// Mitsubishi GX Works2 project: plctest   PLC: Q02/Q02H

PROGRAM MAIN
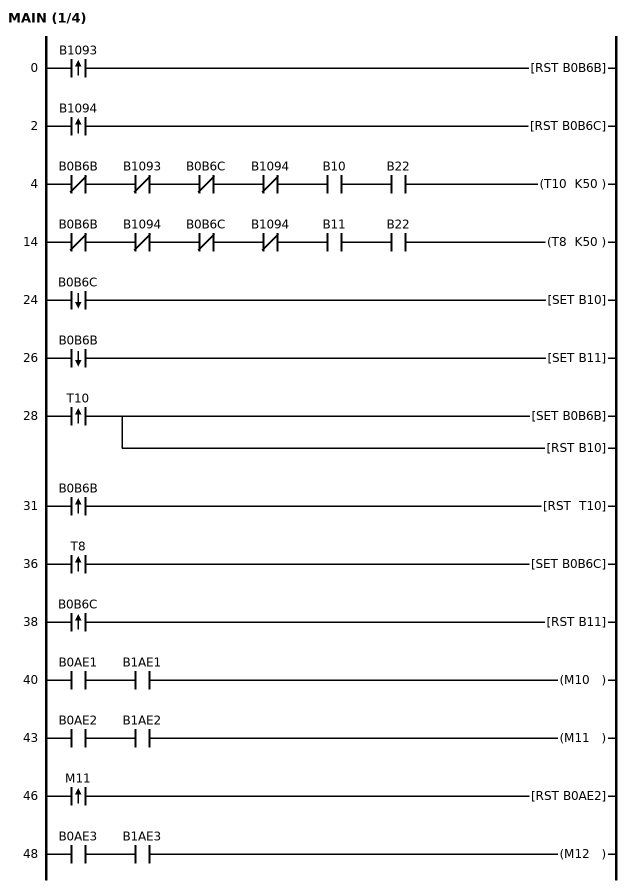
0     LDP     B1093
      RST     B0B6B
2     LDP     B1094
      RST     B0B6C
4     LDI     B0B6B
      ANI     B1093
      ANI     B0B6C
      ANI     B1094
      AND     B10
      AND     B22
      OUT     T10 K50
14    LDI     B0B6B
      ANI     B1094
      ANI     B0B6C
      ANI     B1094
      AND     B11
      AND     B22
      OUT     T8 K50
24    LDF     B0B6C
      SET     B10
26    LDF     B0B6B
      SET     B11
28    LDP     T10
      SET     B0B6B
      RST     B10
31    LDP     B0B6B
      RST     T10
36    LDP     T8
      SET     B0B6C
38    LDP     B0B6C
      RST     B11
40    LD      B0AE1
      AND     B1AE1
      OUT     M10
43    LD      B0AE2
      AND     B1AE2
      OUT     M11
46    LDP     M11
      RST     B0AE2
48    LD      B0AE3
      AND     B1AE3
      OUT     M12
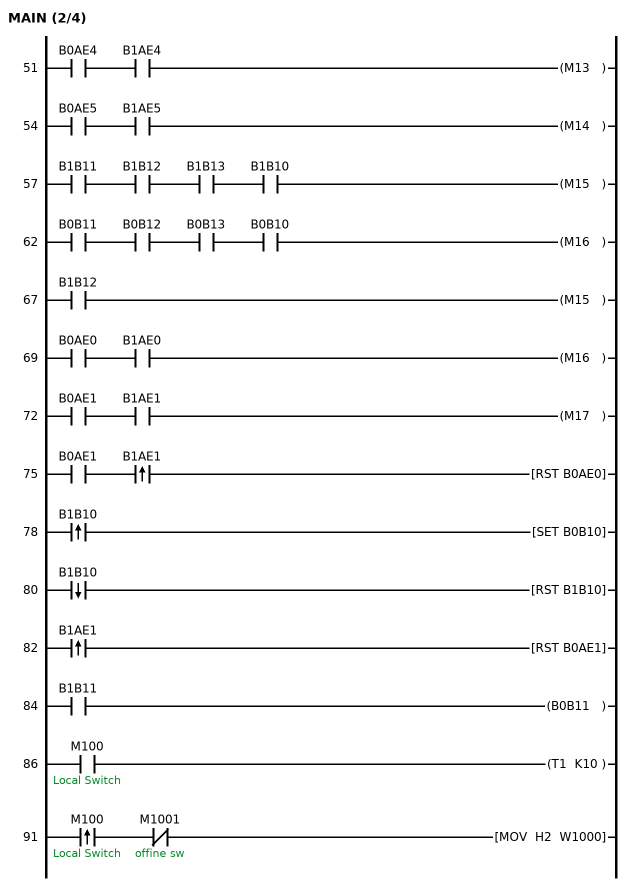
51    LD      B0AE4
      AND     B1AE4
      OUT     M13
54    LD      B0AE5
      AND     B1AE5
      OUT     M14
57    LD      B1B11
      AND     B1B12
      AND     B1B13
      AND     B1B10
      OUT     M15
62    LD      B0B11
      AND     B0B12
      AND     B0B13
      AND     B0B10
      OUT     M16
67    LD      B1B12
      OUT     M15
69    LD      B0AE0
      AND     B1AE0
      OUT     M16
72    LD      B0AE1
      AND     B1AE1
      OUT     M17
75    LD      B0AE1
      ANDP    B1AE1
      RST     B0AE0
78    LDP     B1B10
      SET     B0B10
80    LDF     B1B10
      RST     B1B10
82    LDP     B1AE1
      RST     B0AE1
84    LD      B1B11
      OUT     B0B11
86    LD      M100  ; Local Switch
      OUT     T1 K10
91    LDP     M100  ; Local Switch
      ANI     M1001  ; offine sw
      MOV     H2 W1000
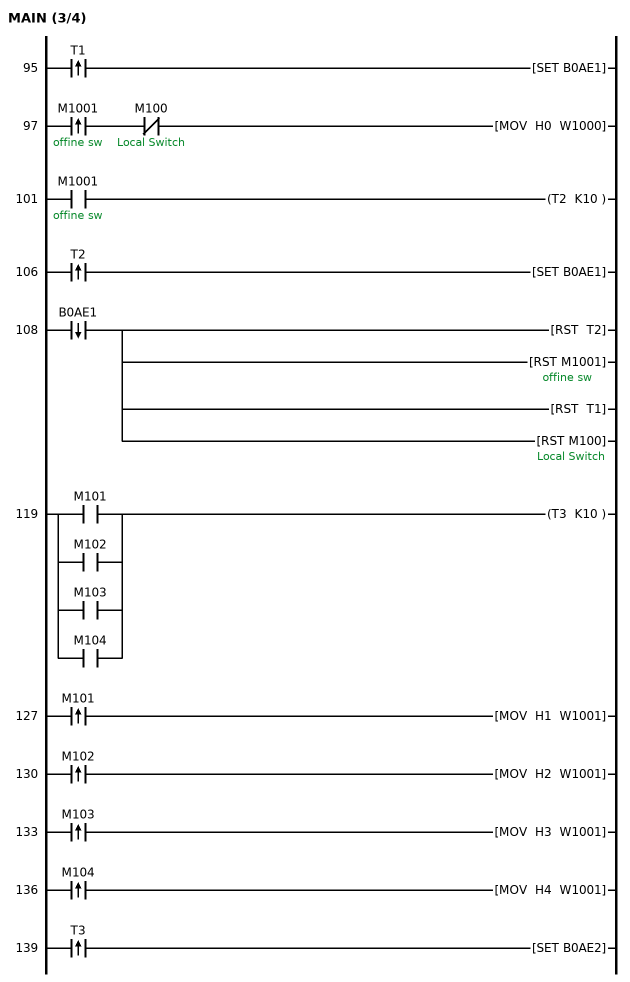
95    LDP     T1
      SET     B0AE1
97    LDP     M1001  ; offine sw
      ANI     M100  ; Local Switch
      MOV     H0 W1000
101   LD      M1001  ; offine sw
      OUT     T2 K10
106   LDP     T2
      SET     B0AE1
108   LDF     B0AE1
      RST     T2
      RST     M1001  ; offine sw
      RST     T1
      RST     M100  ; Local Switch
119   LD      M101
      OR      M102
      OR      M103
      OR      M104
      OUT     T3 K10
127   LDP     M101
      MOV     H1 W1001
130   LDP     M102
      MOV     H2 W1001
133   LDP     M103
      MOV     H3 W1001
136   LDP     M104
      MOV     H4 W1001
139   LDP     T3
      SET     B0AE2
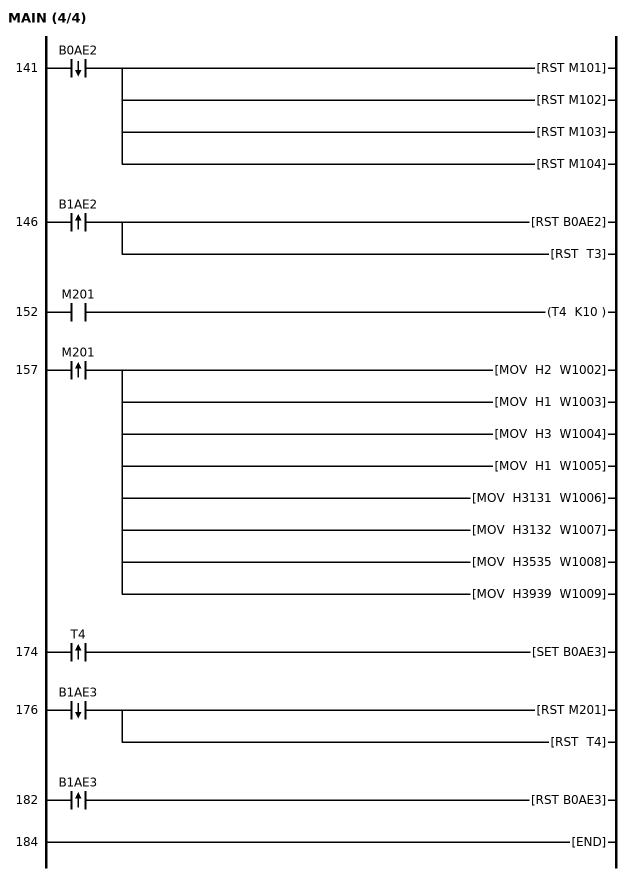
141   LDF     B0AE2
      RST     M101
      RST     M102
      RST     M103
      RST     M104
146   LDP     B1AE2
      RST     B0AE2
      RST     T3
152   LD      M201
      OUT     T4 K10
157   LDP     M201
      MOV     H2 W1002
      MOV     H1 W1003
      MOV     H3 W1004
      MOV     H1 W1005
      MOV     H3131 W1006
      MOV     H3132 W1007
      MOV     H3535 W1008
      MOV     H3939 W1009
174   LDP     T4
      SET     B0AE3
176   LDF     B1AE3
      RST     M201
      RST     T4
182   LDP     B1AE3
      RST     B0AE3
184   END
END_PROGRAM
